{attribute 'qualified_only'}
{attribute 'strict'}
{attribute 'to_string'}
TYPE E_MbRegion :
(
	Auto := 0,
	Coil,
	DiscreteInput,
	InputRegister,
	HoldingRegister
);
END_TYPE

(* stored: Version 1.1.0.1
   DUT E_MbRegion: Id {334fca92-b17e-4248-856f-9d7792218441} *)
